// TIA Portal V16 export
// export: Created 2023-03-29T11:03:44.9340231Z, ExportSetting WithDefaults, DisplayName Totally Integrated Automation Portal, DisplayVersion V16 Update 6, DisplayName TIA Portal Version Control Interface, DisplayVersion V16 Update 2, DisplayName TIA Portal Openness, DisplayVersion V16 Update 6, DisplayName STEP 7 Professional, DisplayVersion V16 Update 6, DisplayName STEP 7 Safety, DisplayVersion V16, DisplayName WinCC Advanced, DisplayVersion V16 Update 6
VAR_GLOBAL   // PLC tag table "Z4"
   Hbit_Auto_Manu_Z4 AT %M16.7 : Bool;
   Hbit_Otwarta_Z4 AT %M16.1 : Bool;
   inputAumagotowośćZ_4 AT %M60.0 : Bool;   // znacznik wejście
   CMD_Awaria_Z_4 AT %M60.7 : Bool;   // Awaria zbiorcza
   setSVMO_Z_4 AT %M60.2 : Bool;   // Znacznik polecenia otwórz w trybie automat
   Hbit_Reset_Z4 AT %M16.6 : Bool;
   inputAumalokalneZ_4 AT %M59.6 : Bool;   // znacznik wejście
   Hbit_Alarm_Z4 AT %M16.0 : Bool;
   inputRuch_Z_4 AT %M59.4 : Bool;
   inputAwariaMomentZ_4 AT %M59.5 : Bool;   // znacznik wejście
   Hbit_Otwórz_Z4 AT %M16.4 : Bool;
   inputAumaautomatZ_4 AT %M59.7 : Bool;   // znacznik wejście
   Hbit_REN_Z4 AT %M16.2 : Bool;
   setAlarm_Moment_Z_4 AT %M60.4 : Bool;   // znacznik alarmu od momentówki w trybie zdalnym (aut/mamnual)
   isGotowość_Z_4 AT %M59.0 : Bool;   // bit gotowości wspólny
   isAUMA_Z_4 AT %M52.5 : Bool;   // przęłącznik wymiany na AUMA
   Hbit_Zamknieta_Z4 AT %M16.3 : Bool;
   inputREMT_Z_4 AT %M59.1 : Bool;   // znacznik wejście zdalne
   Hbit_Zamknij_Z4 AT %M16.5 : Bool;
   inputAumaawariaZ_4 AT %M60.1 : Bool;   // znacznik wejście
   inputOtwartaZ_4 AT %M59.2 : Bool;   // znacznik wejście
   Byte_Status_Z4 AT %MW16 : Word;   // Słowo statusu napędu
   inputZamkniętaZ_4 AT %M59.3 : Bool;   // znacznik wejście
   setSVMC_Z_4 AT %M60.3 : Bool;   // Znacznik polecenia zamknij w trybie automat
   CMD_Close_Z_4 AT %M60.6 : Bool;   // załącz zamykanie
   CMD_Open_Z_4 AT %M60.5 : Bool;   // załącz otwieranie
   edge_Hz_Z4 AT %M92.1 : Bool;   // pamięć zbocza 1 Hz
END_VAR
